{attribute 'enable_dynamic_creation'}
TYPE AdsData :
STRUCT
	description : EventsEnum; //purpose
	
	timestamp : TIMESTRUCT; //relevant timestamp (ex: arrival time)
	
	binaryData : ARRAY[0..100000] OF BYTE; //contents
END_STRUCT
END_TYPE

(* stored: Version 1.1.0.1, ProductVersion 3.1.4024.11
   DUT AdsData: Id {f5237567-f0d5-4783-8173-ee69d89ca101} *)
